TYPE SampleDataStructureLevel2 :
STRUCT
    SampleString : STRING;
    SampleString2 : STRING := '32432423tewtew*-+/';
    SampleInt : INT;
    SampleBool : BOOL;
    SampleBool2 : BOOL := TRUE;
    SampleWString : WSTRING;
    SampleLREAL : LREAL;
END_STRUCT
END_TYPE

(* stored: Version 1.1.0.1, ProductVersion 3.1.4024.9
   DUT SampleDataStructureLevel2: Id {67d1fb94-bf1a-0d94-35ed-7627ad72908c} *)
